FUNCTION_BLOCK SLOT_END_TYPE (* Main loop for simple slot *)
  (* Standard: 61499-2 *)
  (* Version 1.0, 27-05-12, GASR, Universidade do Estado de Santa Catarina *)
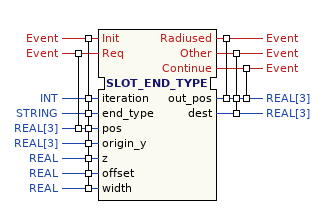
  EVENT_INPUT
    Init WITH iteration, end_type, pos, origin_y, offset, z, width;
    Req WITH pos;
  END_EVENT
  EVENT_OUTPUT
    Radiused WITH out_pos;
    Other WITH out_pos, dest;
    Continue WITH out_pos;
  END_EVENT
  VAR_INPUT
    iteration : INT;
    end_type : STRING;
    pos : ARRAY [0..2] OF REAL;
    origin_y : ARRAY [0..2] OF REAL;
    z : REAL;
    offset : REAL;
    width : REAL;
  END_VAR
  VAR_OUTPUT
    out_pos : ARRAY [0..2] OF REAL;
    dest : ARRAY [0..2] OF REAL;
  END_VAR
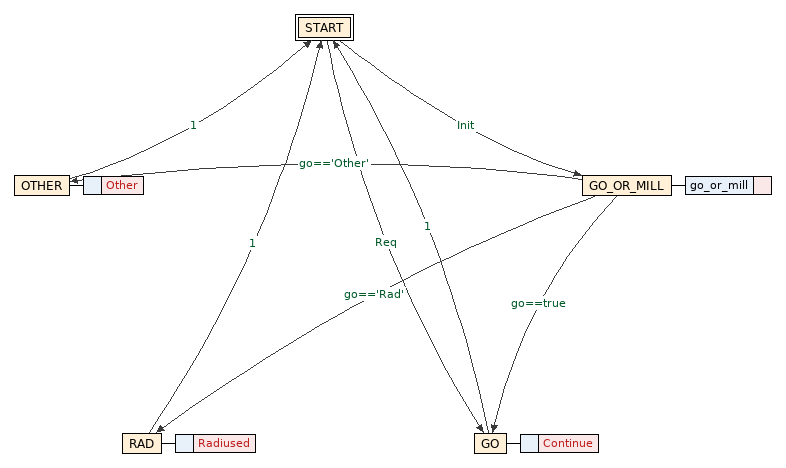
  EC_STATES
    START;
    GO_OR_MILL : go_or_mill;
    GO : -> Continue;
    RAD : -> Radiused;
    OTHER : -> Other;
  END_STATES
  EC_TRANSITIONS
    START TO GO_OR_MILL := Init;
    GO_OR_MILL TO GO := go==true;
    GO_OR_MILL TO RAD := go=='Rad';
    GO_OR_MILL TO OTHER := go=='Other';
    START TO GO := Req;
    GO TO START := 1;
    RAD TO START := 1;
    OTHER TO START := 1;
  END_TRANSITIONS
  ALGORITHM go_or_mill IN Lua:
if( iteration == 1 ) and ( end_type == 'radiused_slot_end_type' ) then
	go = 'Rad'
else
    for i = 1, 2 do
        dest[i] = pos[i] + origin_y[i]*offset*width/2
    end
    dest[3] = z
	go = 'Other'
end
out_pos[1] = pos[1]
out_pos[2] = pos[2]
out_pos[3] = pos[3]
  END_ALGORITHM
END_FUNCTION_BLOCK
(* other elements stored in the file *)
(* VarDeclaration Name=go Type=STRING *)
